(* IEC 61131-3 sources: repolevel_ST_code_completion/output/0121完整版本/repoeval_ProductionLine/readful_result, 6 files *)

(* ---- Motor.st ---- *)
FUNCTION_BLOCK Motor
VAR_INPUT
	MotorI:MotorI;
END_VAR
VAR_OUTPUT
	MotorO:MotorO;
END_VAR
VAR
	WaitTimer: TON;
	InternalSequenceDelay: TIME;
END_VAR

IF MotorI.Overload THEN
	MotorO.FaultStatus := TRUE;
	MotorO.Coil := FALSE;
	RETURN;
END_IF

IF MotorI.ResetFault THEN
	MotorO.FaultStatus := FALSE;
END_IF

IF MotorO.FaultStatus = FALSE THEN
	WaitTimer(IN := TRUE, PT := InternalSequenceDelay);
	IF WaitTimer.Q THEN
		MotorO.Coil := TRUE;
		WaitTimer(IN := FALSE);
	END_IF
ELSE
	MotorO.Coil := FALSE;
END_IF
END_FUNCTION_BLOCK

(* ---- Motor_ResetFault.st ---- *)
METHOD ResetFault : BOOL
VAR_INPUT
	MotorI:MotorI;
END_VAR
VAR_OUTPUT
	MotorO:MotorO;
END_VAR
VAR
	ResetDetect: r_trig;
END_VAR

ResetDetect(CLK := MotorI.FaultReset);

IF ResetDetect.Q THEN
	MotorO.FaultStatus := FALSE;
END_IF

RETURN;
END_OTHER

(* ---- Motor_SetFault.st ---- *)
METHOD SetFault : BOOL
VAR_INPUT
	MotorI:MotorI;
END_VAR
VAR_OUTPUT
	MotorO:MotorO;
END_VAR
VAR
	WaitTimer:TON;
	InternalSequenceDelay:TIME;
END_VAR

IF MotorI.Overload THEN
	MotorO.FaultStatus := TRUE;
	MotorO.Coil := FALSE;
END_IF
END_OTHER

(* ---- Motor_SetWaitTime.st ---- *)
METHOD SetWaitTime : BOOL
VAR_INPUT
	MotorI:MotorI;
	SequenceDelay:TIME;
END_VAR
VAR_OUTPUT
	MotorO:MotorO;
END_VAR
VAR
	WaitTimer:TON;
	InternalSequenceDelay:TIME;
END_VAR

InternalSequenceDelay := SequenceDelay;

IF MotorO.FaultStatus = FALSE THEN
	WaitTimer(IN := TRUE, PT := InternalSequenceDelay);
END_IF

IF WaitTimer.Q THEN
	MotorO.WaitTimeReached := TRUE;
	WaitTimer(IN := FALSE);
	RETURN := TRUE;
ELSE
	MotorO.WaitTimeReached := FALSE;
	RETURN := FALSE;
END_IF
END_OTHER

(* ---- Motor_TurnOff.st ---- *)
METHOD TurnOff : BOOL
VAR_INPUT
	MotorI:MotorI;
END_VAR
VAR_OUTPUT
	MotorO:MotorO;
END_VAR
VAR
	WaitTimer:TON;
	InternalSequenceDelay:TIME;
END_VAR

MotorO.Coil := FALSE;
RETURN;
END_OTHER

(* ---- Motor_TurnOn.st ---- *)
METHOD TurnOn : BOOL
VAR_INPUT
	MotorI:MotorI;
END_VAR
VAR_OUTPUT
	MotorO:MotorO;
END_VAR
VAR
	WaitTimer:TON;
	InternalSequenceDelay:TIME;
END_VAR

IF MotorO.FaultStatus = FALSE THEN
	WaitTimer(IN := TRUE, PT := InternalSequenceDelay);
END_IF

IF WaitTimer.Q THEN
	MotorO.Coil := TRUE;
	WaitTimer(IN := FALSE);
END_IF

RETURN;
END_OTHER
